FUNCTION_BLOCK FB_PM_520x230 EXTENDS FB_PM_Base
//////////////////
// Measurement Solution based on Digiware, but access through PMS Socomec
//////////////////
VAR CONSTANT
	// Characteristics of the object (Same for all instances)
			
END_VAR

VAR_INPUT PERSISTENT
	// Parameters of the Object (instance specific) 
	{attribute 'OPC.UA.DA' := '1'} 
	ParamUnitID					: BYTE := 1 ;									// (NA)unit ID
	ParamInInterfaceSub			: BOOL := TRUE; 								// Serial interface RS422/RS485 TYPE (0:EL6021,1:SUB9)			
END_VAR

VAR_OUTPUT
	//Child objects
	
END_VAR
VAR
	//M_ALARMMANAGEMENT VARIABLES//
	                                                    								
                                                        								

	//M_READ VARIABLES//
		ModbusRTU					: FB_ModbusRTU;								// (NA) FB for Modbus Reading

		MesDataExd				: PM_Standard;								// (NA) Structure of the PM3250
		
		ObjectCom					: INT;										// (NA) Sequence index
									
		Busy						: BOOL;
		StepRead					: UINT;										// (NA) Step for reading 2 blocks of registers
		AX_TrigRead					: ARRAY[1..1] OF R_trig;
		MbStruct					: ARRAY[1..1] OF Struct_InputRTU;	
		MesBlock					: ARRAY[1..1] OF ARRAY[1..120] OF WORD;	
		AX_Addr						: ARRAY[1..1] OF UINT 	:= [19000];
		AX_Qty						: ARRAY[1..1] OF UINT	:= [86];
		AX_UnitId					: ARRAY[1..1] OF BYTE	:= [1];
		AX_Function					: ARRAY[1..1] OF UINT	:= [4];	
		AX_Priority					: ARRAY[1..1] OF UINT	:= [1];
		KK							: INT;
		ComError 					: BOOL;
	//M_INIT VARIABLES //
		OutFBCompleteted			: BOOL;
	// M_EXECUTE VARIABLES //
		
                              

 
END_VAR

METHOD M_AlarmManagement
//////////////////
// Digiware measurement tool alarm and warning management
/////////////////

VAR 
	// Method local variables (reinitialized at each cycle) 
	FB_AlarmCodeManager			: FB_AlarmCodeManager ; 
	
	KK							: BYTE ;		// For loop
	
	CMWarning					: BOOL;			// At least one Digiware device in Alarm
	CMAlarm						: BOOL;			// At least one Digiware device in Alarm
	
END_VAR
//ComError 	:= MbStruct[1].OutError^;
	
TON_ComAlarm(IN:= ComError , PT:= ParamTempoComAlarm, Q=>MesDataExd.MesData.MesAlarmCom) ;	
TON_ComWarning(IN:= ComError  , PT:= ParamTempoComAlarm, Q=>MesWarningCom) ;	

//					General com alarm : All the read FB fucked up


// ALARM CODE //
	FB_AlarmCodeManager(
		bAlarm1			:= MesDataExd.MesData.MesAlarmCom  , 					// Communication Alarm #COM
		bAlarm2			:=FALSE, 		// 
		bAlarm3			:=FALSE, 		// 
		bAlarm4			:=FALSE, 		// 
		bAlarm5			:=FALSE, //
		bAlarm6			:=FALSE, //
		bAlarm7			:=FALSE, //
		bAlarm8			:=FALSE, //
		bAlarm9			:=FALSE, //
		bAlarm10		:=FALSE, //
		bAlarm11		:=FALSE, //
		bAlarm12		:=FALSE, //
		bAlarm13		:=FALSE, //
		bAlarm14		:=FALSE, //
		bAlarm15		:= FALSE , 			// 			 
		wAlarmCode		=>MesDataExd.MesData.MesAlarmCode);

// WARNING CODE //
	FB_AlarmCodeManager(		
		bAlarm1			:=MesWarningCom	,				 // Communication Warning #COM
		bAlarm2			:=FALSE, 		// 
		bAlarm3			:=FALSE, 		// 
		bAlarm4			:=FALSE, 		// 
		bAlarm5			:=FALSE, //
		bAlarm6			:=FALSE, //
		bAlarm7			:=FALSE, //
		bAlarm8			:=FALSE, //
		bAlarm9			:=FALSE, //
		bAlarm10		:=FALSE, //
		bAlarm11		:=FALSE, //
		bAlarm12		:=FALSE, //
		bAlarm13		:=FALSE, //
		bAlarm14		:=FALSE, //
		bAlarm15		:=FALSE, //
		wAlarmCode		=>MesDataExd.MesData.MesWarningCode);		

// EVENT CODE //
END_METHOD

METHOD M_Evaluate : BOOL
VAR_INPUT
END_VAR
END_METHOD

METHOD M_Execute
//////////////////
//  Method Calls 
/////////////////
VAR 
	// Method local variables (reinitialized at each cycle) 
	// EMULATOR
		Psoltot		: REAL;		// Total Solar Power . 
		KK			: BYTE;		// For Loop
	
END_VAR
// READING AND WRITING CLOCK //
	TP1(IN:=NOT TP1.Q , PT:= ParamClockReadTime);
	ClockRead 		:= TP1.Q;

// PERMANENT CONDITIONS //
	MesCP_Read 					:= TRUE  ; 
	
// METHODS CALLS //
	IF bInit THEN
		M_Init() ; 
		bInit					:= FALSE ; 
		
	END_IF

	M_Read() ; 
	
// EMULATOR COM READ  /////////////
	
	
	////////////////////
	M_AlarmManagement();
END_METHOD

METHOD M_Init
VAR 

END_VAR
//Modbus RTU Relay
FOR KK := 1 TO 1 DO 
	MbStruct[KK].InBuffer 		:= ADR(MesBlock[KK]);
	MbStruct[KK].InFunction 	:= AX_Function[KK];
	MbStruct[KK].InQuantity 	:= AX_Qty[KK];
	MbStruct[KK].InStartAddr 	:= AX_Addr[KK];
	MbStruct[KK].InUnitID 		:= AX_UnitId[KK];
	
END_FOR
END_METHOD

METHOD M_Read
//////////////////
//  Read Modbus Variable for PCS . 
/////////////////
VAR 
	// Method local variables (reinitialized at each cycle) 
	MW 					: FB_MergeWordsToFloat; 
	KK					: BYTE;  						// FOR Loop 

	
END_VAR
// CP-Read / Write 

MesDataExd.MesData.MesCP_Read := MesCP_Read ; 
 

IF MesCP_Read  THEN	

ModbusRTU();


FOR KK := 1 TO 1 DO
	AX_TrigRead[KK](CLK  :=ClockRead) ; // CalLocalTimeStruct.wSecond MOD 5 = 0);
	IF AX_TrigRead[KK].Q THEN
		ModbusRTU.M_AddAction_FIFO(InStruct := MbStruct[KK], InPriority := AX_Priority[KK]);
	END_IF
	MbStruct[KK].OutError			:= ADR(ComError);
END_FOR  
						
// PROPERTIES UPDATE // 
	// Block 1
//MW( WORD_STRONG:= MesBlock_Temp[1][1], 	WORD_WEAK := MesBlock_Temp[1][2],	SIGNED:=TRUE, FIX:=0 , SIZE:=2, VAR_OUT := MesDataExd.MesData.MesI2);
	
MW( WORD_STRONG:= MesBlock[1][1], 	WORD_WEAK := MesBlock[1][2], 	VAR_OUT:= MesDataExd.MesData.MesV1);
MW( WORD_STRONG:= MesBlock[1][3], 	WORD_WEAK := MesBlock[1][4], 	VAR_OUT:= MesDataExd.MesData.MesV2);
MW( WORD_STRONG:= MesBlock[1][5], 	WORD_WEAK := MesBlock[1][6], 	VAR_OUT:= MesDataExd.MesData.MesV3);
MW( WORD_STRONG:= MesBlock[1][7], 	WORD_WEAK := MesBlock[1][8], 	VAR_OUT:= MesDataExd.MesData.MesU12);
MW( WORD_STRONG:= MesBlock[1][9], 	WORD_WEAK := MesBlock[1][10], VAR_OUT:= MesDataExd.MesData.MesU23);
                                                                                
MW( WORD_STRONG:= MesBlock[1][11], 	WORD_WEAK := MesBlock[1][12], VAR_OUT:= MesDataExd.MesData.MesU31);
MW( WORD_STRONG:= MesBlock[1][13], 	WORD_WEAK := MesBlock[1][14], VAR_OUT:= MesDataExd.MesData.MesI1);
MW( WORD_STRONG:= MesBlock[1][15], 	WORD_WEAK := MesBlock[1][16], VAR_OUT:= MesDataExd.MesData.MesI2);
MW( WORD_STRONG:= MesBlock[1][17], 	WORD_WEAK := MesBlock[1][18], VAR_OUT:= MesDataExd.MesData.MesI3);
MW( WORD_STRONG:= MesBlock[1][19], 	WORD_WEAK := MesBlock[1][20], VAR_OUT:= MesDataExd.MesData.MesIN);
MW( WORD_STRONG:= MesBlock[1][21], 	WORD_WEAK := MesBlock[1][22], VAR_OUT:= MesDataExd.MesData.MesP1);
MW( WORD_STRONG:= MesBlock[1][23], 	WORD_WEAK := MesBlock[1][24], VAR_OUT:= MesDataExd.MesData.MesP2);
MW( WORD_STRONG:= MesBlock[1][25], 	WORD_WEAK := MesBlock[1][26], VAR_OUT:= MesDataExd.MesData.MesP3);
                                                                                
MW( WORD_STRONG:= MesBlock[1][27], 	WORD_WEAK := MesBlock[1][28], VAR_OUT:= MesDataExd.MesData.MesP);
MW( WORD_STRONG:= MesBlock[1][35], 	WORD_WEAK := MesBlock[1][36], VAR_OUT:= MesDataExd.MesData.MesS);
MW( WORD_STRONG:= MesBlock[1][43], 	WORD_WEAK := MesBlock[1][44], VAR_OUT:= MesDataExd.MesData.MesQ);

//MW( WORD_STRONG_F:= MesBlock[1][7], 	WORD_WEAK_F := MesBlock[1][8], NUMBER_F= MesDataExd.MesData.MesP);
//MW( WORD_STRONG_F:= MesBlock[1][9], 	WORD_WEAK_F := MesBlock[1][10], NUMBER_F= MesDataExd.MesData.MesQ1);
//MW( WORD_STRONG_F:= MesBlock[1][11], 	WORD_WEAK_F := MesBlock[1][12], NUMBER_F= MesDataExd.MesData.MesQ2);
//MW( WORD_STRONG_F:= MesBlock[1][13], 	WORD_WEAK_F := MesBlock[1][14], NUMBER_F= MesDataExd.MesData.MesQ3);
//MW( WORD_STRONG_F:= MesBlock[1][15], 	WORD_WEAK_F := MesBlock[1][16], NUMBER_F= MesDataExd.MesData.MesQ);
//MW( WORD_STRONG_F:= MesBlock[1][23], 	WORD_WEAK_F := MesBlock[1][24], NUMBER_F= MesDataExd.MesData.MesS);

//MW( WORD_STRONG_F:= MesBlock_Temp[4][1], 	WORD_WEAK_F := MesBlock_Temp[4][2], NUMBER_F= MesDataExd.MesData.MesTanPhi);
//MW( WORD_STRONG_F:= MesBlock_Temp[4][3], 	WORD_WEAK_F := MesBlock_Temp[4][4], NUMBER_F= MesDataExd.MesData.MesFreq);
//
//MW( WORD_STRONG_F:= MesBlock_Temp[3][1], 	WORD_WEAK_F := MesBlock_Temp[3][2], NUMBER_F= MesDataExd.MesData.MesEActProd);
//MW( WORD_STRONG_F:= MesBlock_Temp[3][3], 	WORD_WEAK_F := MesBlock_Temp[3][4], NUMBER_F= MesDataExd.MesData.MesEActCons);
//MW( WORD_STRONG_F:= MesBlock_Temp[3][5], 	WORD_WEAK_F := MesBlock_Temp[3][6], NUMBER_F= MesDataExd.MesData.MesEReactProd);
//MW( WORD_STRONG_F:= MesBlock_Temp[3][7], 	WORD_WEAK_F := MesBlock_Temp[3][8], NUMBER_F= MesDataExd.MesData.MesEReactCons);
//MW( WORD_STRONG:= MesBlock_Temp[4][3], 	WORD_WEAK := MesBlock_Temp[4][4],	SIGNED:=TRUE, FIX:=0 , SIZE:=2, VAR_OUT := MesDataExd.MesData.MesFreq);
//MW( WORD_STRONG:= MesBlock_Temp[5][1], 	WORD_WEAK := MesBlock_Temp[5][2],	SIGNED:=TRUE, FIX:=0 , SIZE:=2, VAR_OUT := MesDataExd.MesData.MesEActProd);
//MW( WORD_STRONG:= MesBlock_Temp[5][3], 	WORD_WEAK := MesBlock_Temp[5][4],	SIGNED:=TRUE, FIX:=0 , SIZE:=2, VAR_OUT := MesDataExd.MesData.MesEActCons);
//MW( WORD_STRONG:= MesBlock_Temp[5][5], 	WORD_WEAK := MesBlock_Temp[5][6],	SIGNED:=TRUE, FIX:=0 , SIZE:=2, VAR_OUT := MesDataExd.MesData.MesEReactProd);
//MW( WORD_STRONG:= MesBlock_Temp[5][7], 	WORD_WEAK := MesBlock_Temp[5][8],	SIGNED:=TRUE, FIX:=0 , SIZE:=2, VAR_OUT := MesDataExd.MesData.MesEReactCons);
MesDataExd.Mesdata.MesP	:= MesDataExd.MesData.MesP / 1000.0;
MesDataExd.MesData.MesS	:= MesDataExd.MesData.MesS	/ 1000.0;
MesDataExd.MesData.MesP 	:= -1 * MesDataExd.MesData.MesP;
MesDataExd.MesData.MesP1 	:= -1 * MesDataExd.MesData.MesP1/ 1000.0;
MesDataExd.MesData.MesP2 	:= -1 * MesDataExd.MesData.MesP2/ 1000.0;
MesDataExd.MesData.MesP3 	:= -1 * MesDataExd.MesData.MesP3/ 1000.0;

MesDataExd.MesData.MesQ 	:= -1 * MesDataExd.MesData.MesQ;

MesDataExd.MesData.MesQ 	:= MesDataExd.MesData.MesQ/1000.0;

IF MesDataExd.MesData.MesP <> 0 THEN
MesDataExd.MesData.MesTanPhi := MesDataExd.MesData.MesQ /  MesDataExd.MesData.MesP;

ELSE
MesDataExd.MesData.MesTanPhi := 0;
END_IF



END_IF
END_METHOD

END_FUNCTION_BLOCK

(* stored: Version 1.1.0.1, ProductVersion 3.1.4024.11
   POU FB_PM_520x230: Id {3aa0e0fc-56e2-42c7-bfcd-47ad60c3d338}, SpecialFunc None
   Method M_AlarmManagement: Id {628f34d3-ca6c-42c1-9ad5-f3b2d2730a4e}
   Method M_Evaluate: Id {3f3926a4-c886-4371-803c-f454ed52c04f}
   Method M_Execute: Id {5764c3e6-40a5-4813-ac39-4b0895146822}
   Method M_Init: Id {3c94468d-13ae-4976-b5ce-f428f954b33b}
   Method M_Read: Id {246208a3-5013-4e7b-8c72-bbe18f072b1c} *)
